FUNCTION_BLOCK MixerDepositCheck EXTENDS BaseState
VAR_INPUT
END_VAR
VAR_OUTPUT
END_VAR
VAR
END_VAR

METHOD mIrun : BOOL
IF BasePointer^.MachineFlagsAccessI.pStoring THEN
	RETURN;
ELSE
		mNextState();
END_IF
END_METHOD

END_FUNCTION_BLOCK

(* stored: Version 1.1.0.1, ProductVersion 3.1.4024.12
   POU MixerDepositCheck: Id {934eddb0-057b-43a6-a4ff-f563ff1f33e4}, SpecialFunc None
   Method mIrun: Id {a0114492-1fc8-4577-86d0-76ddba577705} *)
